FUNCTION_BLOCK FB_EMS_HS
VAR_INPUT
END_VAR
VAR_OUTPUT
END_VAR
VAR
// ModBus data structures
	uRead			: U_EMS_HS_Read;
	uWrite			: U_EMS_HS_Write;
	
	// Modbus reading
	tonMBRead		: TON;		// Timer to handle reading requests from device
	fbMBRead		: Tc2_ModbusSrv.FB_MBReadRegs;	// FB for reading modbus register(s)
	bMBRead_Busy	: BOOL;
	bMBRead_Error	: BOOL;
	nMBRead_ErrorID	: UDINT;
	cbMBRead_Read	: UDINT;
	trigMBReadError	: R_TRIG;
	fbGetReadTime	: NT_GetTime;
	trigReadDone	: F_TRIG;
	tsLastRead		: TIMESTRUCT;
	iReads			: UINT;
	iErrorReads		: UINT;

// Modbus writing
	tonMBWrite		: TON;		// Timer to handle writing requests to device
	fbMBWrite		: Tc2_ModbusSrv.FB_MBWriteRegs;	// FB for writing modbus register(s)
	bMBWrite_Busy	: BOOL;
	bMBWrite_Error	: BOOL;
	nMBWrite_ErrorID: UDINT;
	trigWriteDone	: F_TRIG;
	trigMBWriteError: R_TRIG;
	fbGetWriteTime	: NT_GetTime;
	tsLastWrite		: TIMESTRUCT;
	iWrites			: UINT;
	iErrorWrites	: UINT;
	
//Local vars
	bAbortLocal 	: BOOL;
	bManualLocal	: BOOL;
	bProductionLocal: BOOL;
// Simulation
	bSimMode		: BOOL;	// TRUE if simulation should be used (no start device, no setpoints to device)
END_VAR
VAR PERSISTENT
	sIPAddr			: STRING(15);	// Station IP address
	tTimeout		: TIME := T#5S;
END_VAR


// Simulation mode ?
// Only perform communication if NOT in simulation mode
IF (NOT M_Simulation()) THEN

	// Device controller
	M_ModBusRead(	rInterval := 1,
					wAddress := 2501,
					wNoOfRegisters := 23,
					pbDestAddress := ADR(uRead.aWords),
					dwDestSize := SIZEOF(uRead.aWords)	);
	
	M_ModBusWrite(	rInterval := 1, 
					wAddress := 2601,
					wNoOfRegisters := 8,	
					pbSrcAddress := ADR(uWrite.aWords),
					dwSrcSize := SIZEOF(uWrite.aWords)	);
END_IF

// Local state changes
IF (uRead.stVars.eMachStatus = E_EMS_HS_Status.ALARM) THEN
	bAbortLocal := TRUE;
ELSIF (uRead.stVars.stStates.ALARM_IN_PROGRESS) THEN
	bAbortLocal := TRUE;
ELSIF (NOT uRead.stVars.stStates.REMOTE_MODE) THEN
	bAbortLocal := TRUE;
ELSE
	bAbortLocal := FALSE;
END_IF
IF (NOT uRead.stVars.stStates.REMOTE_MODE) THEN
	bManualLocal := TRUE;
	bProductionLocal := FALSE;
ELSE
	bProductionLocal := TRUE;
	bManualLocal := FALSE;
END_IF

METHOD PROTECTED M_CmdNeutral : BOOL
VAR_INPUT
END_VAR
uWrite.stVars.stCommands.REMOTE_START := FALSE;
uWrite.stVars.stCommands.REMOTE_STOP := FALSE;
END_METHOD

METHOD PROTECTED M_Cmdreset : BOOL
VAR_INPUT
END_VAR
END_METHOD

METHOD PROTECTED M_CmdStart : BOOL
VAR_INPUT
END_VAR
uWrite.stVars.stCommands.REMOTE_START := TRUE;
uWrite.stVars.stCommands.REMOTE_STOP := FALSE;
END_METHOD

METHOD PROTECTED M_CmdStop : BOOL
VAR_INPUT
END_VAR
uWrite.stVars.stCommands.REMOTE_START := FALSE;
uWrite.stVars.stCommands.REMOTE_STOP := TRUE;
END_METHOD

/// Read modbus TCP register(s)
METHOD PROTECTED M_ModBusRead : BOOL
VAR_INPUT
	rInterval		: REAL;
	wAddress		: WORD;				// Register address to read
	wNoOfRegisters	: WORD;				// Register to read from station
	pbDestAddress	: POINTER TO BYTE;	// Address of mem to place read data
	dwDestSize		: DWORD;			// Size of mem to place read data
END_VAR
// Timer
tonMBRead(	IN := NOT tonMBRead.Q,
			PT := REAL_TO_TIME(rInterval * 1000.0),
			Q => 	);

// Read data from device via. modbus TCP
fbMBRead(	sIPAddr:= sIPAddr, 				// Station IP address
			nTCPPort:= MODBUS_TCP_PORT, 	// Modbus TCP port (normally 502)
			nUnitID:= 1,//16#FF, 			// If a device is addressed directly via TCP/IP, this value must be 16#FF.
			nQuantity:= wNoOfRegisters,		// Number of words (registers) to read 
			nMBAddr:= wAddress - 1,			// Addres of registers to read ( -1 needed ) 
			cbLength:= dwDestSize,			// Contains the max. byte size of the destination buffer. The minimum buffer byte size must be: nQuantity * 2.
			pDestAddr:= pbDestAddress, 		// Address of the destination buffer into which the data are to be read.
			bExecute:= tonMBRead.Q,			// Trig reading
			tTimeout:= tTimeout, 			// States the length of the timeout that may not be exceeded by execution of the ADS command
			bBusy=> bMBRead_Busy, 
			bError=> bMBRead_Error, 
			nErrId=> , 
			cbRead=> cbMBRead_Read);

// Last read time
trigReadDone(CLK := (fbMBRead.bBusy AND NOT fbMBRead.bError));
trigMBReadError(CLK := bMBRead_Error);
IF (trigReadDone.Q) THEN
	iReads := iReads + 1;
END_IF
IF (trigMBReadError.Q) THEN
	iErrorReads := iErrorReads + 1;
	nMBRead_ErrorID := fbMBRead.nErrId;
END_IF
fbGetReadTime(	NETID:= '', 
				START:= trigReadDone.Q,
				TMOUT:= T#5S, 
				BUSY=> , 
				ERR=> , 
				ERRID=> , 
				TIMESTR=> tsLastRead);

// Station communication status
M_ModBusRead := (cbMBRead_Read = wNoOfRegisters * 2);
END_METHOD

/// Writes ModBus TCP registers
METHOD PROTECTED M_ModBusWrite : BOOL
VAR_INPUT
	rInterval		: REAL;
	wAddress		: WORD;				// Register address to write to
	wNoOfRegisters	: WORD;				// Register(s) to write to station
	pbSrcAddress	: POINTER TO BYTE;	// Address of mem to read source data from
	dwSrcSize		: DWORD;			// Size of mem to read source data from
END_VAR
VAR
END_VAR
// Timer
tonMBWrite(	IN := NOT tonMBWrite.Q,
			PT := REAL_TO_TIME(rInterval * 1000.0),
			Q => 	);

// Write data to device via. modbus TCP
fbMBWrite(	sIPAddr:= sIPAddr, 				// Station IP address
			nTCPPort:= MODBUS_TCP_PORT, 	// Modbus TCP port (normally 502)
			nUnitID:= 1,//16#FF, 			// If a device is addressed directly via TCP/IP, this value must be 16#FF.
			nQuantity:= wNoOfRegisters,		// Number of words (registers) to write 
			nMBAddr:= wAddress - 1,			// Addres of registers to write 
			cbLength:= dwSrcSize,			// Contains the max. byte size of the source buffer. The minimum buffer byte size must be: nQuantity * 2.
			pSrcAddr:= pbSrcAddress,	 	// Address of the source buffer from which, the data are read
			bExecute:= tonMBWrite.Q,		// Trig writing 
			tTimeout:= tTimeout, 			// States the length of the timeout that may not be exceeded by execution of the ADS command
			bBusy=> bMBWrite_Busy, 
			bError=> bMBWrite_Error, 
			nErrId=> );

// Last write time
trigWriteDone(CLK := (fbMBWrite.bBusy AND NOT fbMBWrite.bError));
trigMBWriteError(CLK := bMBWrite_Error);
IF (trigWriteDone.Q) THEN
	iWrites := iWrites + 1;
END_IF
IF (trigMBWriteError.Q) THEN
	iErrorWrites := iErrorWrites + 1;
	nMBWrite_ErrorID := fbMBWrite.nErrId;
END_IF
fbGetWriteTime(	NETID:= '', 
				START:= trigWriteDone.Q,
				TMOUT:= T#5S, 
				BUSY=> , 
				ERR=> , 
				ERRID=> , 
				TIMESTR=> tsLastWrite);

// Station communication status
M_ModBusWrite := trigWriteDone.Q;
END_METHOD

METHOD PROTECTED M_Simulation : BOOL
VAR_INPUT
END_VAR

IF (bSimMode) THEN
	// Simulation mode ENABLED

	// Device start command
	IF (uWrite.stVars.stCommands.REMOTE_START) THEN
		// Device states
		uRead.stVars.eMachStatus := E_EMS_HS_Status.READY;
		uRead.stVars.stStates.MACHINE_READY_TO_WORK := TRUE;
		uRead.stVars.stStates.TEMP_START_BELT_REACHED := TRUE;
		uRead.stVars.stStates.TEMP_START_STEAM_REACHED := TRUE;
		uRead.stVars.stStates.MACHINE_IN_STANDBY := FALSE;
		// Device temperature
		uRead.stVars.rActTempVal := uWrite.stVars.rSetTemp;
	ELSE
		// Device states
		uRead.stVars.eMachStatus := E_EMS_HS_Status.STANDBY;
		uRead.stVars.stStates.MACHINE_READY_TO_WORK := FALSE;
		uRead.stVars.stStates.TEMP_START_BELT_REACHED := FALSE;
		uRead.stVars.stStates.TEMP_START_STEAM_REACHED := FALSE;
		uRead.stVars.stStates.MACHINE_IN_STANDBY := TRUE;
	END_IF
	// Temperature setpoint value
	uRead.stVars.rActTempSetpoint := uWrite.stVars.rSetTemp;
	// Steam setpoint value
	uRead.stVars.rActSteamReq := uWrite.stVars.rSetSteamReq;
	// Fan setpoint value
	uRead.stVars.rActFanReq := uWrite.stVars.rSetFanSpeed;
	// Alarms
	uRead.stVars.stAlarms.TEMP_PROBE_FAULT := FALSE;
	uRead.stVars.stAlarms.FAULT_INVERTER := FALSE;
	uRead.stVars.stAlarms.ENERGY_METER_COM_ERROR := FALSE;
	// Device states
	uRead.stVars.stStates.REMOTE_MODE := TRUE;
	uRead.stVars.stStates.ALARM_IN_PROGRESS := FALSE;
	uRead.stVars.stStates.MACHINE_IN_HEATING := FALSE;
	
	M_Simulation := TRUE;

ELSE
	// Simulation mode DISABLED

	M_Simulation := FALSE;

END_IF
END_METHOD

METHOD PROTECTED M_StaAlarm : BOOL
VAR_INPUT
END_VAR
M_StaAlarm := (uRead.stVars.eMachStatus = E_EMS_HS_Status.ALARM);
END_METHOD

METHOD PROTECTED M_StaReady : BOOL
VAR_INPUT
END_VAR
M_StaReady := (uRead.stVars.eMachStatus = E_EMS_HS_Status.READY);
END_METHOD

METHOD PROTECTED M_StaStandby : BOOL
VAR_INPUT
END_VAR
M_StaStandby := (uRead.stVars.eMachStatus = E_EMS_HS_Status.STANDBY);
END_METHOD

PROPERTY PUBLIC P_bSimulationMode : BOOL
GET
P_bSimulationMode := bSimMode;
END_GET
SET
bSimMode := P_bSimulationMode;
END_SET
END_PROPERTY

PROPERTY P_ModbusIPBarrera : STRING
GET
P_ModbusIPBarrera := sIPAddr;
END_GET
SET
sIPAddr := P_ModbusIPBarrera;
END_SET
END_PROPERTY

PROPERTY PUBLIC P_rSetFanSpeed : REAL
SET
uWrite.stVars.rSetFanSpeed := P_rSetFanSpeed;
END_SET
END_PROPERTY

PROPERTY PUBLIC P_rSetSteamReq : REAL
SET
uWrite.stVars.rSetSteamReq := REAL_TO_DINT(P_rSetSteamReq);
END_SET
END_PROPERTY

PROPERTY PUBLIC P_rSetTemp : REAL
SET
uWrite.stVars.rSetTemp := P_rSetTemp;
END_SET
END_PROPERTY

PROPERTY PUBLIC P_stCellCommandData : ST_EMS_HS_Write
GET // PUBLIC
P_stCellCommandData := uWrite.stVars;
END_GET
SET // PUBLIC
uWrite.stVars := P_stCellCommandData;
END_SET
END_PROPERTY

PROPERTY PUBLIC P_stCellStatusData : ST_EMS_HS_Read
GET
P_stCellStatusData := uRead.stVars;
END_GET
END_PROPERTY

END_FUNCTION_BLOCK

(* stored: Version 1.1.0.1, ProductVersion 3.1.4024.5
   POU FB_EMS_HS: Id {1e7d32d3-1fc5-459f-b7ae-c1510d53e863}, SpecialFunc None
   Method M_CmdNeutral: Id {df67d31e-796c-48bf-9279-1a2c3e34719f}
   Method M_Cmdreset: Id {a7d6c347-a00b-4483-9ff7-2f8ac31f3725}
   Method M_CmdStart: Id {f88e3817-dcb4-4b7e-b186-fd80a0644fe2}
   Method M_CmdStop: Id {499747e8-b3b8-4d1d-bd40-dd2916fabc16}
   Method M_ModBusRead: Id {1d805d5b-72cb-4562-b8f3-7b5f95a6d3c6}
   Method M_ModBusWrite: Id {ad7e0026-c981-45e4-82b3-0ad200bde4c2}
   Method M_Simulation: Id {d1d60dd9-27e1-43df-9925-59e6970c9666}
   Method M_StaAlarm: Id {dea6e8a1-5a0d-4fbc-a58a-c08fe03b92da}
   Method M_StaReady: Id {771b0fd9-5c4d-427d-90ca-aa71d928646a}
   Method M_StaStandby: Id {ca89f6b8-7639-45bd-8a53-e6e632c1abd0}
   Property P_bSimulationMode: Id {4e2d2f17-1689-4614-8d3f-7a9b2b482f3e}
   Get Get: Id {746a8707-d105-4e70-875e-58b7822a198d}
   Set Set: Id {c4f43457-4532-4734-a2f4-21feb602d173}
   Property P_ModbusIPBarrera: Id {32e6a03d-bfcb-4215-82a9-1b3613b8830d}
   Get Get: Id {89502621-3507-4af2-87bd-1904daa8e14e}
   Set Set: Id {4cec20f3-52c9-49ff-bae4-4ecbef7b7857}
   Property P_rSetFanSpeed: Id {0f0f0c95-f786-4d61-a94a-c3d5057da639}
   Set Set: Id {87576d72-ef69-45f3-8182-519a042b52f2}
   Property P_rSetSteamReq: Id {5e767a20-e0c3-4191-b6ad-37c4649aa6a5}
   Set Set: Id {b27ff9f6-0783-4737-8f27-f0c33a7008ed}
   Property P_rSetTemp: Id {d7170c0b-2e33-4cea-a6d4-bd60bbf61bce}
   Set Set: Id {0a709314-5109-47c2-9d95-e4df4df9ca64}
   Property P_stCellCommandData: Id {7f055175-13e6-4580-9ad2-b3d43fae28bd}
   Get Get: Id {59dcfd2a-aa1c-4095-8660-27c25adf3c82}
   Set Set: Id {f679871d-679f-4f0a-a06a-c918464db843}
   Property P_stCellStatusData: Id {7a826849-9064-407e-b166-1851ac98572c}
   Get Get: Id {c50d1c87-523f-4925-b7f9-a59866f475e8} *)
